(* 
| :Description: This function block represents basic digital input and can be used for creating an instance of signle digital input device like buttons, switches, sensors.
| To get the current status of digital input use "Value" property. To simulate state of the input by software set "Enable Force" parameter and change value via "MR_ResetForceValue" and "MR_SetForceValue" methods.
*)
FUNCTION_BLOCK FB_DigitalInputExt EXTENDS FB_DigitalInput
VAR
	(* Internal commands *)
	bInit 				: BOOL;		(*  *)
	bAbort				: BOOL;		(*  *)
	bReset				: BOOL;		(*  *)
	bTimeoutTracking	: BOOL;		(* Watchdog timer control bit *)
	
	(* Internal status *)
	bActive				: BOOL;		(*  *)
	bErrorTimedout		: BOOL;		(* Timeout coccured while waiting for signal *)
	eDigitalInputState	: E_DigitalInputExState;
	
	(*Internal parameters*)
	tTimeout			: TIME;		(* Input timeout *)
	bEnableTimeout		: BOOL;		(* Enable using timeout *)
	
	(* Function blocks *)
	bStartWatchdog		: BOOL;
	tonWatchdog			: TON;		(* Input timeout watchdog *)
	
END_VAR

bActive := eDigitalInputState >= DIGITAL_INPUT_EX_IDLE; //OR eDigitalInputState = DIGITAL_INPUT_EX_ABORTING;

StateMachine();

tonWatchdog( IN := bStartWatchdog, PT := tTimeout);

PROPERTY Active : REFERENCE TO BOOL
GET
Active REF= bActive;
END_GET
END_PROPERTY

PROPERTY CurrentTimeout : REFERENCE TO TIME
GET
CurrentTimeout REF= tonWatchdog.ET;
END_GET
END_PROPERTY

PROPERTY EnableTimeout : BOOL
GET
EnableTimeout := bEnableTimeout;
END_GET
SET
bEnableTimeout := EnableTimeout;
END_SET
END_PROPERTY

PROPERTY ErrorTimedout : REFERENCE TO BOOL
GET
ErrorTimedout REF= bErrorTimedout;
END_GET
END_PROPERTY

METHOD MR_Abort : BOOL
VAR_INPUT
END_VAR
IF eDigitalInputState > DIGITAL_INPUT_EX_UNINITIALIZED THEN
	bAbort := TRUE;
	MR_Abort := FALSE;
	eDigitalInputState := DIGITAL_INPUT_EX_ABORTING;
	fbMachineLogger.MR_AddLogs(CONCAT(sName,' : abort requested'));	
	
ELSIF eDigitalInputState = DIGITAL_INPUT_EX_UNINITIALIZED THEN
	bAbort := FALSE;
	MR_Abort := TRUE;
	fbMachineLogger.MR_AddLogs(CONCAT(sName,' : abort done'));	
	
END_IF
END_METHOD

METHOD MR_FirstCycleEx : BOOL
VAR_INPUT
	sName			: STRING;
	sModuleType		: STRING;
	sPortID			: STRING;
	bEnableTimeout	: BOOL;
	tDefaultTimeout : TIME;
END_VAR
THIS^.sName := sName;
THIS^.ModuleType := sModuleType;
THIS^.PortID := sPortID;
THIS^.bEnableTimeout := bEnableTimeout;
THIS^.tTimeout := tDefaultTimeout;
END_METHOD

METHOD MR_Init : BOOL
VAR_INPUT
END_VAR
IF eDigitalInputState = DIGITAL_INPUT_EX_UNINITIALIZED THEN
	bInit := TRUE;
	MR_Init := FALSE;
	eDigitalInputState := DIGITAL_INPUT_EX_INITIALIZING;
	fbMachineLogger.MR_AddLogs(CONCAT(sName,' : initialization requested'));		
	
ELSIF eDigitalInputState = DIGITAL_INPUT_EX_IDLE AND bInit THEN
	bInit := FALSE;
	MR_Init := TRUE;
	fbMachineLogger.MR_AddLogs(CONCAT(sName,' : initialization done'));	

END_IF
END_METHOD

METHOD MR_Reset : BOOL
VAR_INPUT
END_VAR
IF eDigitalInputState = DIGITAL_INPUT_EX_IDLE THEN
	bReset := TRUE;
	MR_Reset := FALSE;
	eDigitalInputState := DIGITAL_INPUT_EX_RESET;
	fbMachineLogger.MR_AddLogs(CONCAT(sName,' : reset requested'));	
	
ELSIF eDigitalInputState = DIGITAL_INPUT_EX_RESET_DONE THEN
	bReset := FALSE;
	MR_Reset := TRUE;
	fbMachineLogger.MR_AddLogs(CONCAT(sName,' : reset done'));	
	
END_IF
END_METHOD

METHOD MR_StartTracking
VAR_INPUT
END_VAR
IF eDigitalInputState = DIGITAL_INPUT_EX_IDLE AND bEnableTimeout AND NOT bErrorTimedout THEN
	bTimeoutTracking := TRUE;
	eDigitalInputState := DIGITAL_INPUT_EX_TIMEOUT_TRACKING;
	fbMachineLogger.MR_AddLogs(CONCAT(sName,' : start tracking requested'));	
	
END_IF
END_METHOD

METHOD PROTECTED MS_Abort
VAR_INPUT
END_VAR
eDigitalInputState := DIGITAL_INPUT_EX_UNINITIALIZED;
END_METHOD

METHOD PROTECTED MS_Idle
VAR_INPUT
END_VAR
;
END_METHOD

METHOD PROTECTED MS_Initializing
VAR_INPUT
END_VAR
(* To-Do add alarm declaration *)

eDigitalInputState := DIGITAL_INPUT_EX_READY_INITIALIZED;
END_METHOD

METHOD PROTECTED MS_ReadyInitialized
VAR_INPUT
END_VAR
eDigitalInputState := DIGITAL_INPUT_EX_IDLE;
END_METHOD

METHOD PROTECTED MS_Reset
VAR_INPUT
END_VAR
bErrorTimedout := FALSE;
eDigitalInputState := DIGITAL_INPUT_EX_RESET_DONE;
END_METHOD

METHOD PROTECTED MS_ResetDone
VAR_INPUT
END_VAR
IF NOT bReset THEN
	eDigitalInputState := DIGITAL_INPUT_EX_IDLE;
END_IF
END_METHOD

METHOD PROTECTED MS_TimeoutTracking
VAR_INPUT
END_VAR
IF tonWatchdog.Q THEN
	(* To-Do raise alarm *)
	bErrorTimedout := TRUE;
	bStartWatchdog := FALSE;
	eDigitalInputState := DIGITAL_INPUT_EX_TIMEOUT_TRACKING_DONE;
	
ELSE
	bStartWatchdog := TRUE;
	
	IF bRisingTrigger OR bFallingTrigger THEN
		bStartWatchdog := FALSE;
		eDigitalInputState := DIGITAL_INPUT_EX_TIMEOUT_TRACKING_DONE;
	
	END_IF
END_IF
END_METHOD

METHOD PROTECTED MS_TimeoutTrackingDone
VAR_INPUT
END_VAR
bTimeoutTracking := FALSE;
eDigitalInputState := DIGITAL_INPUT_EX_IDLE;
END_METHOD

METHOD PROTECTED MS_Uninitialized
VAR_INPUT
END_VAR
bInit := FALSE;
bAbort := FALSE;
bReset := FALSE;
bTimeoutTracking := FALSE;

bRisingTrigger := FALSE;
bFallingTrigger := FALSE;
bErrorTimedout := FALSE;

tonWatchdog( IN := FALSE, PT := tTimeout);
END_METHOD

PROPERTY State : REFERENCE TO E_DigitalInputExState
GET
State REF= eDigitalInputState;
END_GET
END_PROPERTY

METHOD PROTECTED StateMachine
VAR_INPUT
END_VAR
CASE eDigitalInputState OF
	DIGITAL_INPUT_EX_UNINITIALIZED:
		MS_Uninitialized();
		
	DIGITAL_INPUT_EX_INITIALIZING:
		MS_Initializing();
		
	DIGITAL_INPUT_EX_READY_INITIALIZED:
		MS_ReadyInitialized();
		
	DIGITAL_INPUT_EX_IDLE:
		MS_Idle();
		
	DIGITAL_INPUT_EX_TIMEOUT_TRACKING:
		MS_TimeoutTracking();	
	
	DIGITAL_INPUT_EX_TIMEOUT_TRACKING_DONE:
		MS_TimeoutTrackingDone();	
	
	DIGITAL_INPUT_EX_RESET:
		MS_Reset();

	DIGITAL_INPUT_EX_RESET_DONE:
		MS_ResetDone();
	
	DIGITAL_INPUT_EX_ABORTING:
		MS_Abort();
	
END_CASE
END_METHOD

PROPERTY Timeout : TIME
GET
Timeout := tTimeout;
END_GET
SET
tTimeout := Timeout;
END_SET
END_PROPERTY

END_FUNCTION_BLOCK

(* stored: Version 1.1.0.1, ProductVersion 3.1.4024.12
   POU FB_DigitalInputExt: Id {306ccf3b-f75f-4f5a-aaf1-3bc1695862ee}, SpecialFunc None
   Folder FirstCycle: Id {59b9490c-7564-40d9-a364-72728a7381e1}
   Folder Properties: Id {4fb8016b-45e3-4a3d-b371-fb412110d960}
   Folder Parameters: Id {ba1b78c9-38d1-4d81-ac75-ca573a6c21f8}
   Folder Status: Id {9884cd86-cd9d-4e6a-aa7c-f6b34f67e1a8}
   Folder Requests: Id {df908729-3267-471e-b430-98fdc99dbb68}
   Folder StateMachine: Id {98cf4a4b-af28-43a7-a816-5488f5ecc4bf}
   Property Active: Id {1d1a69cd-28d9-423d-bb74-e76a3e7ed21b}
   Get Get: Id {aa7c41af-7747-4fa0-ab55-76a819e5e66e}
   Property CurrentTimeout: Id {22a807fe-3288-4153-be59-dda883612369}
   Get Get: Id {0e4ea362-8db8-4615-b141-e09995c1bf4c}
   Property EnableTimeout: Id {c464567b-8c3a-4926-92e7-604757f82f4c}
   Get Get: Id {3208d6b6-29dc-4051-ad73-50179b7f05e9}
   Set Set: Id {91a99842-bfc5-4f26-9d2c-6668b9100653}
   Property ErrorTimedout: Id {1be3e029-3bca-407c-937c-f0f88a10cbb6}
   Get Get: Id {d2a095c7-8b0c-4bdf-bb76-1241bcf74fb6}
   Method MR_Abort: Id {d651dbff-bcc4-40dd-8d44-714051fee34c}
   Method MR_FirstCycleEx: Id {b46e9c86-8a6c-43e2-8e5c-b65700dd99fb}
   Method MR_Init: Id {249ec19e-ac72-499e-867d-a64e2e632d55}
   Method MR_Reset: Id {371b7467-c075-42d9-9418-b309d2dc3eba}
   Method MR_StartTracking: Id {75e4d076-6bab-4670-86b7-2ec7acfe7812}
   Method MS_Abort: Id {06d43a0e-1b62-4f03-849e-b216dbee1c7d}
   Method MS_Idle: Id {c9021290-8628-4719-99cd-3a17835336c7}
   Method MS_Initializing: Id {b055f464-a013-4d48-95a1-158f75cf165e}
   Method MS_ReadyInitialized: Id {1b61816b-0e7c-4697-9ca3-c03e6bd5d600}
   Method MS_Reset: Id {f205e94c-98e3-4fb9-8a08-802b6d6f0588}
   Method MS_ResetDone: Id {715f7b19-a107-4bf8-9568-8b18f6f174b1}
   Method MS_TimeoutTracking: Id {0c54f001-4e07-4807-ab06-00c535c96c31}
   Method MS_TimeoutTrackingDone: Id {11d2a47d-c948-40af-89e8-f42aed2dc73e}
   Method MS_Uninitialized: Id {c4cd865c-a5ab-41c3-9123-fb0902cdecc1}
   Property State: Id {f2f07911-aff7-4060-9993-1e2879f7a7de}
   Get Get: Id {2e9c72ec-1f76-49d1-a6de-5249c865d093}
   Method StateMachine: Id {861b9bc6-6819-49a9-b962-25af74d19c71}
   Property Timeout: Id {d91bde1a-1044-46b4-b6ec-d9553838fd7e}
   Get Get: Id {983c364e-6ad9-4042-8429-aaa5e8aa1a02}
   Set Set: Id {bcd9be63-53f1-4333-b660-1f59e098930c} *)
